PROGRAM OP30_Error
VAR
	OP30_Step_Err_1: TON;
	OP30_Step_Err_2: TON;
	OP30_Step_Err_3: TON;
	OP30_Step_Err_4: TON;
	OP30_Step_Err_5: TON;
	OP30_Step_Err_6: TON;
END_VAR


// Set ERROR ACTIVE
IF ((OP30_GVL.OP30_ErrorWord_0<>0) OR (OP30_GVL.OP30_ErrorWord_1<>0) OR (OP30_GVL.OP30_ErrorWord_2<>0)) THEN
	OP30_GVL.OP30_ErrorActive:= TRUE;
END_IF

//Reset ErrorActive
IF (OP30_GVL.OP30_HMI_Reset) THEN 
	OP30_GVL.OP30_ErrorActive:= FALSE;
	OP30_GVL.OP30_ErrorWord_0:= 0;
	OP30_GVL.OP30_ErrorWord_1:= 0;
	OP30_GVL.OP30_ErrorWord_2:= 0;	
END_IF

// Auto Seq Step Error

//Horizontal Servo is not in home or safe-work position 
OP30_Step_Err_1(IN:=(OP30_GVL.OP30_AutoSeq=70) , PT:=T#5S , Q=> , ET=> );
IF (OP30_GVL.OP30_AutoSeq=70 AND OP30_Step_Err_1.Q) THEN
	OP30_GVL.OP30_ErrorWord_0.0:=TRUE;
END_IF


//Horizontal Servo not reaching pick position 
OP30_Step_Err_1(IN:=(OP30_GVL.OP30_AutoSeq=80) , PT:=T#5S , Q=> , ET=> );
IF (OP30_GVL.OP30_AutoSeq=80 AND NOT OP30_HORI_SERVO_ON_WRK_PICK AND OP30_Step_Err_1.Q) THEN
	OP30_GVL.OP30_ErrorWord_0.1:=TRUE;
END_IF

// Gripper is not closing
OP30_Step_Err_2(IN:=OP30_GVL.OP30_AutoSeq=82 , PT:=T#5S , Q=> , ET=> );
IF (OP30_GVL.OP30_AutoSeq=82 AND OP30_Step_Err_2.Q) THEN
	OP30_GVL.OP30_ErrorWord_0.2:=TRUE;
END_IF

// Vertical Servo not reaching work position 
OP30_Step_Err_3(IN:=OP30_GVL.OP30_AutoSeq=100 , PT:=T#5S , Q=> , ET=> );
IF (OP30_GVL.OP30_AutoSeq=100 AND OP30_Step_Err_3.Q) THEN
	OP30_GVL.OP30_ErrorWord_0.3:=TRUE;
END_IF

// Vertical Servo not reaching safe-work position 
OP30_Step_Err_3(IN:=OP30_GVL.OP30_AutoSeq=130 , PT:=T#5S , Q=> , ET=> );
IF (OP30_GVL.OP30_AutoSeq=130 AND OP30_Step_Err_3.Q) THEN
	OP30_GVL.OP30_ErrorWord_0.4:=TRUE;
END_IF

// Checking the gripper condition is opened or not
OP30_Step_Err_3(IN:=OP30_GVL.OP30_AutoSeq=140 , PT:=T#5S , Q=> , ET=> );
IF (OP30_GVL.OP30_AutoSeq=140 AND OP30_Step_Err_3.Q) THEN
	OP30_GVL.OP30_ErrorWord_0.5:=TRUE;
END_IF

//  Horizontal sevo not moving to place position
OP30_Step_Err_3(IN:=OP30_GVL.OP30_AutoSeq=160 , PT:=T#5S , Q=> , ET=> );
IF (OP30_GVL.OP30_AutoSeq=160 AND OP30_Step_Err_3.Q) THEN
	OP30_GVL.OP30_ErrorWord_0.6:=TRUE;
END_IF

//  Vertical sevo not moving to place position
OP30_Step_Err_3(IN:=OP30_GVL.OP30_AutoSeq=180 , PT:=T#5S , Q=> , ET=> );
IF (OP30_GVL.OP30_AutoSeq=180 AND OP30_Step_Err_3.Q) THEN
	OP30_GVL.OP30_ErrorWord_0.7:=TRUE;
END_IF

// Vertical Servo not reaching safe-work position 
OP30_Step_Err_3(IN:=OP30_GVL.OP30_AutoSeq=210 , PT:=T#5S , Q=> , ET=> );
IF (OP30_GVL.OP30_AutoSeq=210 AND OP30_Step_Err_3.Q) THEN
	OP30_GVL.OP30_ErrorWord_0.8:=TRUE;
END_IF

//  Horizontal sevo not moving to safe work position
OP30_Step_Err_3(IN:=OP30_GVL.OP30_AutoSeq=240 , PT:=T#5S , Q=> , ET=> );
IF (OP30_GVL.OP30_AutoSeq=240 AND OP30_Step_Err_3.Q) THEN
	OP30_GVL.OP30_ErrorWord_0.9:=TRUE;
END_IF

END_PROGRAM

(* stored: Version 1.1.0.1, ProductVersion 3.1.4024.11
   POU OP30_Error: Id {f6587571-ca84-4826-b15e-3c0fac18ed1d}, SpecialFunc None *)
